TYPE QualityInspectionComSubscribe :
STRUCT
  Request : QualityInspectionComRequest; // contains booleans that are used to start a specific sequence.
  Equipment : QualityInspectionComSubscribeEquipment;  // structs for equipment objects which are used by the bridges
END_STRUCT
END_TYPE

(* stored: Version 1.1.0.1
   DUT QualityInspectionComSubscribe: Id {32dcc99d-8773-4ce4-b0c3-8590347035c1} *)
